FUNCTION_BLOCK xPPU_PicAlpha
VAR_INPUT
	i_error: POINTER TO ErrorManager;
	i_process: POINTER TO ProcessManager;
	i_state: POINTER TO StateTracker;
END_VAR
VAR
	m_emptyParams: ParameterSet;
	m_subRes: EOperationResult;
END_VAR

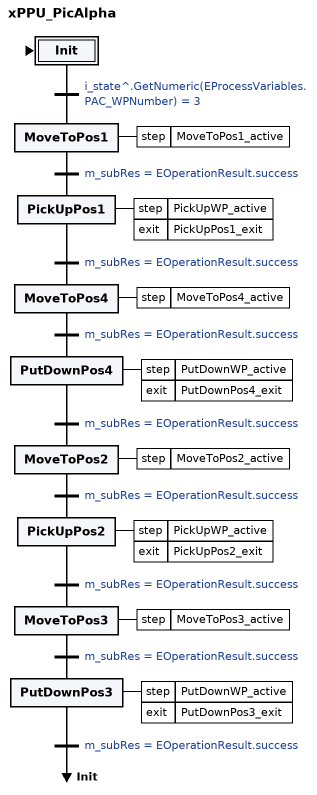
INITIAL_STEP Init:
END_STEP
TRANSITION FROM Init TO MoveToPos1
    := i_state^.GetNumeric(EProcessVariables.PAC_WPNumber) = 3;
END_TRANSITION
STEP MoveToPos1:
    MoveToPos1_active(N);  // step action
END_STEP
TRANSITION FROM MoveToPos1 TO PickUpPos1
    := m_subRes = EOperationResult.success;
END_TRANSITION
STEP PickUpPos1:
    PickUpWP_active(N);  // step action
    PickUpPos1_exit(P0);  // exit action
END_STEP
TRANSITION FROM PickUpPos1 TO MoveToPos4
    := m_subRes = EOperationResult.success;
END_TRANSITION
STEP MoveToPos4:
    MoveToPos4_active(N);  // step action
END_STEP
TRANSITION FROM MoveToPos4 TO PutDownPos4
    := m_subRes = EOperationResult.success;
END_TRANSITION
STEP PutDownPos4:
    PutDownWP_active(N);  // step action
    PutDownPos4_exit(P0);  // exit action
END_STEP
TRANSITION FROM PutDownPos4 TO MoveToPos2
    := m_subRes = EOperationResult.success;
END_TRANSITION
STEP MoveToPos2:
    MoveToPos2_active(N);  // step action
END_STEP
TRANSITION FROM MoveToPos2 TO PickUpPos2
    := m_subRes = EOperationResult.success;
END_TRANSITION
STEP PickUpPos2:
    PickUpWP_active(N);  // step action
    PickUpPos2_exit(P0);  // exit action
END_STEP
TRANSITION FROM PickUpPos2 TO MoveToPos3
    := m_subRes = EOperationResult.success;
END_TRANSITION
STEP MoveToPos3:
    MoveToPos3_active(N);  // step action
END_STEP
TRANSITION FROM MoveToPos3 TO PutDownPos3
    := m_subRes = EOperationResult.success;
END_TRANSITION
STEP PutDownPos3:
    PutDownWP_active(N);  // step action
    PutDownPos3_exit(P0);  // exit action
END_STEP
TRANSITION FROM PutDownPos3 TO Init
    := m_subRes = EOperationResult.success;
END_TRANSITION

ACTION MoveToPos1_active:
m_subRes := i_process^.Execute(
	EBehaviorType.control_primitive,
	EPrimitives.PicAlpha_MoveToPos1,
	m_emptyParams);
END_ACTION

ACTION MoveToPos2_active:
m_subRes := i_process^.Execute(
	EBehaviorType.control_primitive,
	EPrimitives.PicAlpha_MoveToPos2,
	m_emptyParams);
END_ACTION

ACTION MoveToPos3_active:
m_subRes := i_process^.Execute(
	EBehaviorType.control_primitive,
	EPrimitives.PicAlpha_MoveToPos3,
	m_emptyParams);
END_ACTION

ACTION MoveToPos4_active:
m_subRes := i_process^.Execute(
	EBehaviorType.control_primitive,
	EPrimitives.PicAlpha_MoveToPos4,
	m_emptyParams);
END_ACTION

ACTION PickUpPos1_exit:
i_state^.ShiftProduct(EProducts.PAC_product2, EProducts.PicAlpha_product);
i_state^.ShiftProduct(EProducts.PAC_product3, EProducts.PAC_product2);
END_ACTION

ACTION PickUpPos2_exit:
i_state^.ShiftProduct(EProducts.PAC_product2, EProducts.PicAlpha_product);
END_ACTION

ACTION PickUpWP_active:
m_subRes := i_process^.Execute(
	EBehaviorType.control_primitive,
	EPrimitives.PicAlpha_PickUpWP,
	m_emptyParams);
END_ACTION

ACTION PutDownPos3_exit:
i_state^.ShiftProduct(EProducts.PicAlpha_product, EProducts.PAC_product2);
END_ACTION

ACTION PutDownPos4_exit:
//shift product from PicAlpha to SSC
i_state^.ShiftProduct(EProducts.PicAlpha_product, EProducts.SSC_product1);
END_ACTION

ACTION PutDownWP_active:
m_subRes := i_process^.Execute(
	EBehaviorType.control_primitive,
	EPrimitives.PicAlpha_PutDownWp,
	m_emptyParams);
END_ACTION

END_FUNCTION_BLOCK

(* stored: Version 1.1.0.1, ProductVersion 3.1.4024.4
   POU xPPU_PicAlpha: Id {5176e747-510f-403f-81f7-57cd8dd0c8c2}, SpecialFunc None
   Action MoveToPos1_active: Id {a0991c78-5824-4ef2-8fa8-4456e4d1a45e}
   Action MoveToPos2_active: Id {6a91b0dc-0544-46c8-ba12-917fd6d76d70}
   Action MoveToPos3_active: Id {224e64d2-c26b-408a-8cf2-2e2a5aa28ae0}
   Action MoveToPos4_active: Id {72bbdb3c-e1ad-4e87-9599-21e42bfea0b4}
   Action PickUpPos1_exit: Id {eefb59a3-8cdb-4c84-84b4-ab43ba38956f}
   Action PickUpPos2_exit: Id {b8c0b797-8ee4-497f-b643-cf0043fb6892}
   Action PickUpWP_active: Id {58463b08-495e-495a-9b02-cf0843842b47}
   Action PutDownPos3_exit: Id {0ba6192f-3d98-42f2-a35f-a5994e6f2937}
   Action PutDownPos4_exit: Id {4b97a5b5-346a-48a6-a790-3a3dd7480d7f}
   Action PutDownWP_active: Id {72766da6-2c09-4527-a8c9-928e1dd61436} *)
